Omron CX-Programmer project NewProject (CX-Programmer 9.75)

# PLC OMRON: CP1E N30

## Global symbols (name address type ; comment)
T000 BOOL  ; T0
T001 BOOL  ; T1
T002 BOOL  ; T2

## Program NewProgram1 (cyclic task 0)
Local symbols
Green1 100.01 BOOL  ; 100.01
Green2 100.02 BOOL  ; 100.02
M1 10.01 BOOL  ; 10.01
M2 10.02 BOOL  ; 10.02
M3 10.03 BOOL  ; 10.03
M4 10.04 BOOL  ; 10.04
MPS 100.00 BOOL  ; 100.00
PNP 0.00 BOOL  ; 0.00
Red1 100.05 BOOL  ; 100.05
Red2 100.06 BOOL  ; 100.06
Stop 0.01 BOOL  ; 0.01
Sw1 0.02 BOOL  ; 0.02
Sw2 0.03 BOOL  ; 0.03
Sw3 0.04 BOOL  ; 0.04
Sw4 0.05 BOOL  ; 0.05
Yellow1 100.03 BOOL  ; 100.03
Yellow2 100.04 BOOL  ; 100.04
Yellow3 100.07 BOOL  ; 100.07

### Section Section1

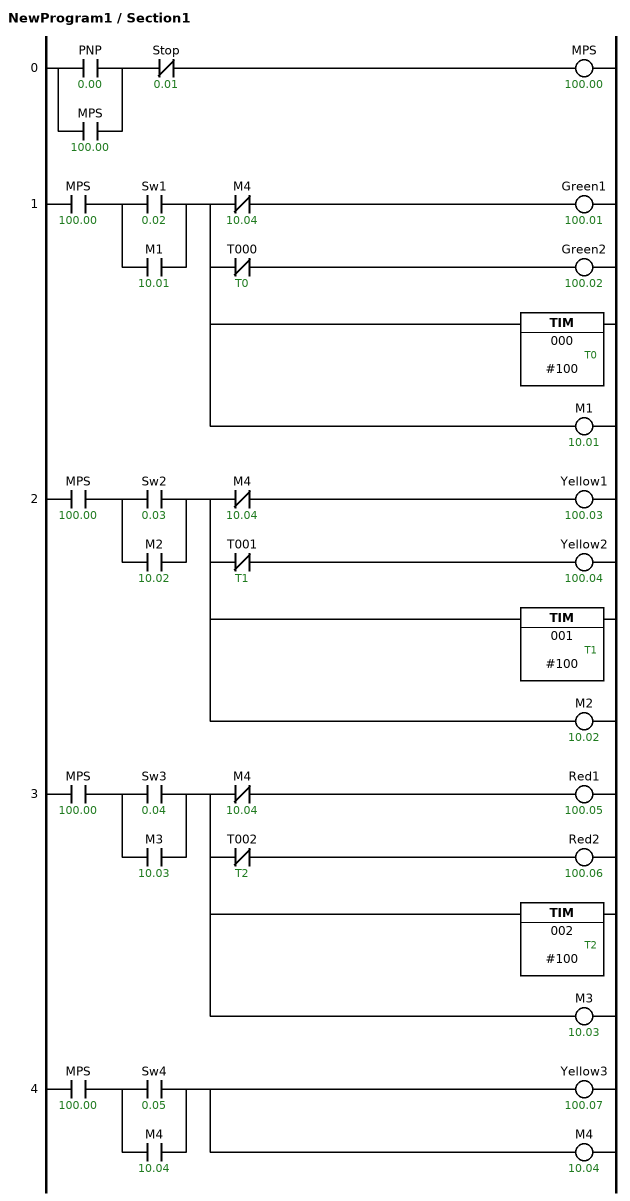
; rung 0
LD PNP  ; 0.00
OR MPS  ; 100.00
ANDNOT Stop  ; 0.01
OUT MPS  ; 100.00
; rung 1
LD MPS  ; 100.00
LD Sw1  ; 0.02
OR M1  ; 10.01
ANDLD
OUT TR0
ANDNOT M4  ; 10.04
OUT Green1  ; 100.01
LD TR0
ANDNOT T000  ; T0
OUT Green2  ; 100.02
LD TR0
TIM 000 #100  ; T0
OUT M1  ; 10.01
; rung 2
LD MPS  ; 100.00
LD Sw2  ; 0.03
OR M2  ; 10.02
ANDLD
OUT TR0
ANDNOT M4  ; 10.04
OUT Yellow1  ; 100.03
LD TR0
ANDNOT T001  ; T1
OUT Yellow2  ; 100.04
LD TR0
TIM 001 #100  ; T1
OUT M2  ; 10.02
; rung 3
LD MPS  ; 100.00
LD Sw3  ; 0.04
OR M3  ; 10.03
ANDLD
OUT TR0
ANDNOT M4  ; 10.04
OUT Red1  ; 100.05
LD TR0
ANDNOT T002  ; T2
OUT Red2  ; 100.06
LD TR0
TIM 002 #100  ; T2
OUT M3  ; 10.03
; rung 4
LD MPS  ; 100.00
LD Sw4  ; 0.05
OR M4  ; 10.04
ANDLD
OUT Yellow3  ; 100.07
OUT M4  ; 10.04

### Section END
; rung 0
END(001)